INTERFACE I_InputPorts

METHOD PUBLIC Accept
VAR_INPUT
	Visitor : I_InputPortVisitor;
END_VAR
END_METHOD

METHOD PUBLIC AddDataAsInputPort : I_InputPort
VAR_INPUT
	Name : T_MAXSTRING;
	Data : I_Datatype;
END_VAR
END_METHOD

METHOD AddInputPort
VAR_INPUT
	InputPort : I_InputPort;
END_VAR
END_METHOD

METHOD PUBLIC TryGetInputPortByName : BOOL
VAR_INPUT
	Name : T_MAXSTRING;
	Destination : REFERENCE TO I_InputPort;
END_VAR
END_METHOD

END_INTERFACE

(* stored: Version 1.1.0.1, ProductVersion 3.1.4024.12
   Itf I_InputPorts: Id {71bbf865-1e29-4075-b9c2-e305690245b8}
   Method Accept: Id {65e9e350-b4da-4b31-beb2-b7dd75c935ea}
   Method AddDataAsInputPort: Id {fa5250ab-a88e-4b57-81f9-a513fe6d8457}
   Method AddInputPort: Id {e9138a76-36f7-41c8-9618-e82fbbae5526}
   Method TryGetInputPortByName: Id {03568ac7-b326-418d-92c6-36ccec2fe85b} *)
